TYPE (* Typedef of the ISO CF/user information data structure *)
  (* Version 1.0, 2025-09-04, Franz Höpfinger, initial API and implementation and/or initial documentation *)
  PACKAGE isobus::pgn;
  IMPORT eclipse4diac::core::TypeHash;
  IMPORT isobus::pgn::HANDLE::UNVALID;
  IMPORT isobus::pgn::ADDRESS::NULL_A;
  IMPORT isobus::pgn::USERFUNC_e::undefined;
  CF_INFO_T : STRUCT
    s16Handle : INT := UNVALID; (* Network member handle of the CF / user *)
    u8SourceAddress : BYTE := NULL_A; (* Source address (SA) of the control function (CF) / user *)
    u8CanIdx : BYTE; (* CAN-Bus node / index of the control function (CF) / user *)
    au8Name : isobus::pgn::CF_NAME_T; (* CF ISOBUS NAME *)
    eIsoUserFunct : SINT := undefined; (* Internal used CF function type *)
    bExternalCf : BOOL; (* External CF on the CAN network *)
    bIsAnnounced : BOOL; (* ISO_TRUE if the CF is active and full announced *)
    bIsActive : BOOL; (* NIU specific: ISO_TRUE if the CF is not in an error state or logged off *)
  END_STRUCT;
END_TYPE
